(* PLC project CoDeSys External Library Template, WAGO e!COCKPIT e!COCKPIT, author 3S - Smart Software Solutions GmbH *)
(* stored: creationDateTime 2019-10-29T12:37:19.776809, version 3.5.5.30, modificationDateTime 2019-10-29T12:36:39.3744516, organization 3S - Smart Software Solutions GmbH *)
(* Library project template with all possible element types, docu and a sample project structure *)

FUNCTION fnCRC16Walidacja : BOOL
  VAR_INPUT
    sKomunikat : alSTRINGKomunikat;
    wCRC16Wynik : WORD;
  END_VAR
  VAR
    wCRC16_modbus : WORD;
    intPetla : INT;
    arwTelegram : ARRAY[1..512] OF BYTE;
  END_VAR

            wCRC16_modbus := fnCRC16Obliczanie(sKomunikat);

IF wCRC16_modbus = wCRC16Wynik THEN
	fnCRC16Walidacja := TRUE;
	ELSE	
	fnCRC16Walidacja := FALSE;
END_IF

          
END_FUNCTION
